(* IEC 61131-3 sources: StringExt/src/Ar/StringExt, 3 files *)

(* ---- StringExt.typ ---- *)
(*
 * File: StringExt.typ
 * Copyright (c) 2023 Loupe
 * https://loupe.team
 *
 * This file is part of StringExt, licensed under the MIT License.
 *
 *)

TYPE
	STREXT_ERR_enum :
		(
		STREXT_ERR_BUFFER_TOO_SMALL := -4, (*Destination buffer is too small for the result*)
		STREXT_ERR_RANGE := -3, (*Value does not fit in the destination type*)
		STREXT_ERR_INVALID_FORMAT := -2, (*String is not a valid literal of the expected form*)
		STREXT_ERR_INVALID_INPUT := -1
		);
	STREXT_HEXPREFIX_enum :
		(
		STREXT_HEXPREFIX_NONE := 0, (*FF*)
		STREXT_HEXPREFIX_0X, (*0xFF*)
		STREXT_HEXPREFIX_IEC, (*16#FF*)
		STREXT_HEXPREFIX_DOLLAR (*$FF*)
		);
	StrExtArgs_typ : 	STRUCT  (*Arguments for formatter*)
		r : ARRAY[0..4]OF REAL; (*Reals*)
		s : ARRAY[0..4]OF UDINT; (*Pointers to String*)
		b : ARRAY[0..4]OF BOOL; (*Booleans*)
		i : ARRAY[0..4]OF DINT; (*Signed Integers*)
	END_STRUCT;
END_TYPE

(* ---- StringExt.fun ---- *)
(*
 * File: StringExt.fun
 * Copyright (c) 2023 Loupe
 * https://loupe.team
 *
 * This file is part of StringExt, licensed under the MIT License.
 *
 *)

FUNCTION lstrip : UDINT (*Strips the leading characters from a string*)
	VAR_INPUT
		pString : UDINT;
		pChars : UDINT;
	END_VAR
END_FUNCTION

FUNCTION rstrip : UDINT (*Strips the trailing characters from a string*)
	VAR_INPUT
		pString : UDINT;
		pChars : UDINT;
	END_VAR
END_FUNCTION

FUNCTION atoui : UDINT (*Converts a string to a UDINT value, allowing values greater than the DINT maximum*)
	VAR_INPUT
		pString : UDINT;
	END_VAR
END_FUNCTION

FUNCTION uitoa : UDINT (*Converts a UDINT to a string, allowing values greater than the DINT maximum*)
	VAR_INPUT
		Value : UDINT;
		pString : UDINT;
	END_VAR
END_FUNCTION

FUNCTION ByteToHexString : UDINT (*Converts bytes to a hex string*)
	VAR_INPUT
		pByte : UDINT;
		NumBytes : UDINT;
		pString : UDINT;
	END_VAR
END_FUNCTION

FUNCTION HexStringToDINT : DINT (*Converts a Hex String to a DINT*) (*$GROUP=User,$CAT=User,$GROUPICON=User.png,$CATICON=User.png*)
	VAR_INPUT
		pHexStr : UDINT;
	END_VAR
END_FUNCTION

FUNCTION HexStringToUDINT : DINT (*Parses a hex string with an optional 0x, 16# or $ prefix. Returns 0 on success or a STREXT_ERR_enum value; the parsed value is written through pValue*) (*$GROUP=User,$CAT=User,$GROUPICON=User.png,$CATICON=User.png*)
	VAR_INPUT
		pHexStr : UDINT; (*Pointer to the string to parse*)
		pValue : UDINT; (*Pointer to the UDINT that receives the value*)
	END_VAR
END_FUNCTION

FUNCTION UDINTToHexString : DINT (*Formats a UDINT as a hex string. Returns the string length or a STREXT_ERR_enum value*) (*$GROUP=User,$CAT=User,$GROUPICON=User.png,$CATICON=User.png*)
	VAR_INPUT
		Value : UDINT; (*Value to format*)
		pString : UDINT; (*Pointer to the destination buffer*)
		Size : UDINT; (*Size of the destination buffer, including the terminator*)
		NumDigits : USINT; (*Zero pad to this many digits, 1..8. 0 for the shortest representation*)
		Prefix : USINT; (*Notation to use, see STREXT_HEXPREFIX_enum*)
	END_VAR
END_FUNCTION

FUNCTION GenerateTimestampMS_1 : UINT (*Generate a time stamp string from a DTStructure variable*)
	VAR_INPUT
		pDTStructure : UDINT;
		pTimestamp : UDINT;
		TimestampLength : UDINT;
	END_VAR
END_FUNCTION

FUNCTION GenerateTimestampMS : UINT (*Generate a time stamp string from a DTStructure variable*)
	VAR_INPUT
		pDTStructure : UDINT;
		pTimestamp : UDINT;
		TimestampLength : UDINT;
	END_VAR
END_FUNCTION

FUNCTION GenerateTimestamp : UINT (*Generate a time stamp string from a DATE_AND_TIME variable*)
	VAR_INPUT
		DT1 : DATE_AND_TIME;
		pTimestamp : UDINT;
		TimestampLength : UDINT;
	END_VAR
END_FUNCTION

FUNCTION strncat4 : UINT (*Combine strings pSource1 through pSource4 into pDest, with ' / ' between source strings*) (*$GROUP=User*)
	VAR_INPUT
		pDest : UDINT;
		pSource1 : UDINT;
		pSource2 : UDINT;
		pSource3 : UDINT;
		pSource4 : UDINT;
		MaxLength : UDINT;
	END_VAR
END_FUNCTION

FUNCTION ToUpper : UDINT (*Converts a string to upper case*) (*$GROUP=User*)
	VAR_INPUT
		pString : UDINT;
	END_VAR
END_FUNCTION

FUNCTION ToLower : UDINT (*Converts a string to lower case*) (*$GROUP=User*)
	VAR_INPUT
		pString : UDINT;
	END_VAR
END_FUNCTION

FUNCTION Timestamp_TO_DT : DATE_AND_TIME
	VAR_INPUT
		pDT : UDINT;
		pTimestamp : UDINT;
	END_VAR
END_FUNCTION

FUNCTION appendArrayIndex : UDINT (*Appends [Value] to string*) (*$GROUP=User,$CAT=User,$GROUPICON=User.png,$CATICON=User.png*)
	VAR_INPUT
		Value : UDINT;
		pString : UDINT;
	END_VAR
END_FUNCTION

FUNCTION SplitFileName : UDINT (*Seperates file extension from file name*) (*$GROUP=User,$CAT=User,$GROUPICON=User.png,$CATICON=User.png*)
	VAR_INPUT
		pFileName : UDINT; (*Pointer to the string containing file name and extension*)
		pName : UDINT; (*Pointer to location to copy file name (optional)*)
		pExtension : UDINT; (*Pointer to location to copy extension (optional)*)
	END_VAR
END_FUNCTION

FUNCTION stringlcpy : UDINT (*Copies strings safely*)
	VAR_INPUT
		pDest : UDINT;
		pSrc : UDINT;
		dSize : UDINT;
	END_VAR
END_FUNCTION

FUNCTION stringlcat : UDINT (*Concats strings safely*)
	VAR_INPUT
		pDest : UDINT;
		pSrc : UDINT;
		dSize : UDINT;
	END_VAR
END_FUNCTION

FUNCTION string2wstring : UDINT (*Converts String to WString*)
	VAR_INPUT
		pDest : UDINT; (*Pointer to String where contents will be copied*)
		pSrc : UDINT; (*Pointer to WString of contents to be converted*)
		dSize : UDINT; (*Size of destination String*)
	END_VAR
END_FUNCTION

FUNCTION wstring2string : UDINT (*Converts Wstring to String*)
	VAR_INPUT
		pDest : UDINT; (*Pointer to WString where contents will be copied*)
		pSrc : UDINT; (*Pointer to String of contents to be converted*)
		dSize : UDINT; (*Size of destination WString*)
	END_VAR
END_FUNCTION

FUNCTION char2wchar : UINT (*Converts Char to WChar*)
	VAR_INPUT
		character : USINT; (*Char to be converted*)
	END_VAR
END_FUNCTION

FUNCTION wchar2char : USINT (*Converts WChar to Char*)
	VAR_INPUT
		wcharacter : UINT; (*WChar to be converted*)
	END_VAR
END_FUNCTION

FUNCTION formatString : DINT (*Safe fromat string similar to sprintf*)
	VAR_INPUT
		dest : STRING[80]; (*Destination of formatted string*)
		destSize : UDINT; (*Size of destination*)
		format : STRING[80]; (*String with formatters*)
		pArgs : StrExtArgs_typ; (*Pointer to argument structure*)
	END_VAR
END_FUNCTION

FUNCTION stringfTime : UDINT (*Format time to string*)
	VAR_INPUT
		dest : UDINT; (*Pointer to destination*)
		destSize : UDINT; (*Size of destination*)
		format : UDINT; (*Format to use*)
		time : DATE_AND_TIME; (*Time to format*)
	END_VAR
END_FUNCTION

FUNCTION stringpTime : DATE_AND_TIME (*Parse time string*)
	VAR_INPUT
		src : UDINT; (*String to parse*)
		format : UDINT; (*Assumed format of time string*)
	END_VAR
END_FUNCTION

FUNCTION stringdtoa : UDINT
	VAR_INPUT
		value : LREAL;
		buffer : STRING[80];
		ndigits : UDINT;
		bufferSize : UDINT;
	END_VAR
END_FUNCTION

FUNCTION stringftoa : UDINT
	VAR_INPUT
		value : REAL;
		buffer : STRING[80];
		ndigits : UDINT;
		bufferSize : UDINT;
	END_VAR
END_FUNCTION

FUNCTION stringstrtod : LREAL
	VAR_INPUT
		value : STRING[80];
		pEnd : REFERENCE TO STRING[80];
	END_VAR
END_FUNCTION

FUNCTION stringstrtof : REAL
	VAR_INPUT
		value : STRING[80];
		pEnd : REFERENCE TO STRING[80];
	END_VAR
END_FUNCTION

(* ---- StringExt.var ---- *)
(*
 * File: StringExt.var
 * Copyright (c) 2023 Loupe
 * https://loupe.team
 *
 * This file is part of StringExt, licensed under the MIT License.
 *
 *)
VAR CONSTANT
	STREXT_INVALID_CHAR : USINT := 221;
	STREXT_MAX_UDINT : UDINT := 4294967295;
END_VAR
